(* CODESYS project DUT.ecp

Project tree, tasks and I/O mapping:
  PFC200_CS_2ETH_RS_CAN_DPS : 750-8212 PFC200 2ETH RS, WAGO, order no. 0750-8212, version 5.14.3.63
    application Application
      libraries: 
      task PLC_Task (cyclic, interval t#10ms, priority 14) calls PLC_PRG
      data type MyMotor
      program Traditional_Declaration [ST]
      program PLC_PRG [ST]
    Kbus : Kbus, WAGO, version 1.4.0.2
        unmapped channels: K-BUS diagnostics
    MODBUS
      MODBUS : MODBUS, WAGO, order no. n/a, version 1.1.1.15
    Serial
      COM1 : COM1, WAGO, version 0.0.0.19
    Common.PCI
  libraries: VisuSymbols, 3.5.8.0 (System); WagoVisuIcons, 1.0.0.7 (WAGO)
  text list GlobalTextList
*)

// PFC200_CS_2ETH_RS_CAN_DPS/Application/MyMotor
TYPE MyMotor :
STRUCT
	sMotorName : STRING(20);
	xMotor_on_off : BOOL;
	xFault : BOOL;
	rMotor_Voltage: REAL;
	rMotor_Current : REAL;
END_STRUCT
END_TYPE

// PFC200_CS_2ETH_RS_CAN_DPS/Application/PLC_PRG
PROGRAM PLC_PRG
VAR
	aMotors : ARRAY[1..MaxMotors] OF MyMotor;
	i : INT;
	xMotorProblems : BOOL;
END_VAR

VAR CONSTANT
	MaxMotors: BYTE := 4;
END_VAR

// Add fixed simulation values

//Motor1
	aMotors[1].sMotorName:= 'Pump 1'; 
	aMotors[1].xMotor_on_off := TRUE;
	aMotors[1].xFault := FALSE;
	aMotors[1].rMotor_Voltage:= 230.4;
	aMotors[1].rMotor_Current := 1.3;
	
//Motor2
	aMotors[2].sMotorName := 'Pump 2'; 
	aMotors[2].xMotor_on_off := TRUE;
	aMotors[2].xFault := TRUE;
	aMotors[2].rMotor_Voltage:= 228.9;
	aMotors[2].rMotor_Current := 1.2;


//Motor3
	aMotors[3].sMotorName := 'Pump 3'; 
	aMotors[3].xMotor_on_off := TRUE;
	aMotors[3].xFault:= FALSE;
	aMotors[3].rMotor_Voltage := 231.2;
	aMotors[3].rMotor_Current := 1.35;
	
	
// For loop to check if 1 of the motors is in fault.
//The variable xMotorProblems should will not be resettet automatically in this example	
	FOR i := 1 TO MaxMotors DO
		IF aMotors[i].xFault = TRUE THEN
			xMotorProblems := TRUE;
		END_IF
	END_FOR

END_PROGRAM

// PFC200_CS_2ETH_RS_CAN_DPS/Application/Traditional_Declaration
PROGRAM Traditional_Declaration
VAR
	sMotorName_1 : STRING(20);
	xMotor_on_off_1 : BOOL;
	xFault_1 : BOOL;
	rMotor_Voltage_1: REAL;
	rMotor_Current_1 : REAL;
	
	sMotorName_2 : STRING(20);
	xMotor_on_off_2 : BOOL;
	xFault_2 : BOOL;
	rMotor_Voltage_2: REAL;
	rMotor_Current_2 : REAL;
	
	sMotorName_3 : STRING(20);
	xMotor_on_off_3 : BOOL;
	xFault_3 : BOOL;
	rMotor_Voltage_3: REAL;
	rMotor_Current_3 : REAL;
END_VAR

// Add fixed simulation values

//Motor1
	sMotorName_1 := 'Pump 1'; 
	xMotor_on_off_1 := TRUE;
	xFault_1 := FALSE;
	rMotor_Voltage_1:= 230.4;
	rMotor_Current_1 := 1.3;
	
//Motor2
	sMotorName_2 := 'Pump 2'; 
	xMotor_on_off_2 := TRUE;
	xFault_2 := TRUE;
	rMotor_Voltage_2:= 228.9;
	rMotor_Current_2 := 1.2;


//Motor3
	sMotorName_3 := 'Pump 3'; 
	xMotor_on_off_3 := TRUE;
	xFault_3 := FALSE;
	rMotor_Voltage_3:= 231.2;
	rMotor_Current_3 := 1.35;

END_PROGRAM
